Staubli VAL3: getMenu.pgx

public program getMenu(string& x_sMenu[], bool& x_bUseMenu[])
// set the function button using the menu string
  local num i
begin
  //
  // STAUBLI Application
  // set the x_bUseMenu using the Menu
  // array string
  //
  for i=0 to (size(x_bUseMenu)-1)
    x_bUseMenu[i]=false
    if (size(x_sMenu)-1)>=i
      if x_sMenu[i]!=""
        // active the button
        x_bUseMenu[i]=true
      endIf
    endIf
  endFor
end
